VAR_GLOBAL
	{attribute 'OPC.UA.DA':='1'}
	{attribute 'OPC.UA.DA.Access':='1'}
	I AT %I*: ARRAY[0..7] OF BOOL;
	
	{attribute 'OPC.UA.DA':='1'}
	{attribute 'OPC.UA.DA.Access':='1'}
	Q AT %Q*: ARRAY[0..7] OF BOOL;
END_VAR

(* stored: Version 1.1.0.1, ProductVersion 3.1.4024.12
   GVL gIO: Id {b502dacf-f837-4a1a-9176-5415efc890a4} *)
